{attribute 'GeneratedUsingTerminal: EK1100-0000-0018'}
{attribute addProperty BoxType "EK1100-0000-0018"}
{attribute addProperty Id "Beckhoff_EK13xxEK1122Beckhoff_EK13xxEK1122_1E36FC7A8A_0003_EK1322_0000_0017EK1322_0DA715C26A_0002_EK1310_0000_0017EK1310_0DA715C26"}
{attribute addProperty CRC "3747626250"}
{attribute addProperty Size "20"}
TYPE Beckhoff_EK13xx_DF603D0A EXTENDS EK1100_AB5A9467 :
STRUCT
	{attribute addProperty Name "Beckhoff_EK13xxEK1122"}
	{attribute addProperty PreviousPort "Beckhoff EK13xx : B"}
	Beckhoff_EK13xxEK1122 : Beckhoff_EK13xxEK1122_1E36FC7A;
	{attribute addProperty Name "A_0003_EK1322_0000_0017"}
	{attribute addProperty PreviousPort "Beckhoff EK13xxEK1122 : C"}
	A_0003_EK1322_0000_0017 : EK1322_0DA715C2;
	{attribute addProperty Name "A_0002_EK1310_0000_0017"}
	{attribute addProperty PreviousPort "A_0003(EK1322-0000-0017) : C"}
	A_0002_EK1310_0000_0017 : EK1310_0DA715C2;
END_STRUCT
END_TYPE

(* stored: Version 1.2.0.0, ProductVersion 3.1.4024.9
   DUT Beckhoff_EK13xx_DF603D0A: Id {b9b8ad52-087a-4c6a-9dc0-9ad8683b6de7} *)
